// TIA Portal project "Project3_Sequence_Command" (V18)

(* hardware
DEVICE "S7-1500/ET200MP station_1"  S7-1500 station
   slot 0: "Rail_0"  Rack  6ES7 590-1***0-0AA0
DEVICE "S7-1500/ET200MP station_2"  S7-1500 station
   slot 0: "PM 190W 120/230VAC"  PM 190W 120/230VAC  6EP1333-4BA00
   slot 0: "Rail_0"  Rack  6ES7 590-1***0-0AA0
   slot 1: "PLC_1"  CPU 1516-3 PN/DP  6ES7 516-3AN01-0AB0  V2.1
      slot 3: "CPU display_1"  6ES7591-1BA00-0AA0
      slot 32768: "PROFINET interface_1"  X1
         slot 32769: "Port_1"  X1 P1
         slot 32770: "Port_2"  X1 P2
      slot 33024: "PROFINET interface_2"  X2
         slot 33025: "Port_1"  X2 P1
      slot 33280: "DP interface_1"  X3
   slot 2: "DI 32x24VDC HF_1"  DI 32x24VDC HF  6ES7 521-1BL00-0AB0  V2.2
   slot 3: "DQ 32x24VDC/0.5A HF_1"  DQ 32x24VDC/0.5A HF  6ES7 522-1BL01-0AB0  V1.1
   slot 4: "AI 8xU/R/RTD/TC HF_1"  AI 8xU/R/RTD/TC HF  6ES7 531-7PF00-0AB0  V1.1
   slot 5: "AQ 4xU/I HF_1"  AQ 4xU/I HF  6ES7 532-5ND00-0AB0  V1.1
*)

// ===== PLC "PLC_1"  CPU 1516-3 PN/DP =====

VAR_GLOBAL   // PLC tag table "Default tag table"
   "Tag_1" AT %I0.0 : Bool;
   "Tag_2" AT %Q0.0 : Bool;
   "Tag_3" AT %I0.1 : Bool;
   "Tag_4" AT %Q0.1 : Bool;
   "Tag_5" AT %M0.0 : Bool;
   "Tag_6" AT %Q0.2 : Bool;
   "Tag_7" AT %I0.2 : Bool;
   "Tag_8" AT %I0.3 : Bool;
   "Tag_9" AT %M1.0 : Bool;
   "Tag_10" AT %M1.1 : Bool;
   "Tag_11" AT %M0.1 : Bool;
   "Tag_12" AT %M0.2 : Bool;
   "Tag_13" AT %M1.2 : Bool;
   "Tag_14" AT %MD0 : Time;
   "Tag_15" AT %MD4 : Time;
   "Tag_16" AT %MD8 : Time;
   "Tag_17" AT %MD12 : Time;
   "Tag_18" AT %MD16 : Time;
   "Tag_19" AT %MW0 : Int;
   "Tag_20" AT %M1.3 : Bool;
   "Tag_21" AT %M2.0 : Bool;
END_VAR

// folder: System blocks/Program resources

DATA_BLOCK "DB1"   // DB1
{ S7_Optimized_Access := 'TRUE' }
AUTHOR : Simatic
FAMILY : IEC
NAME : IEC_TMR
VERSION : 1.0
// stored: InstanceOfName IEC_TIMER
"IEC_TIMER"
BEGIN
END_DATA_BLOCK

DATA_BLOCK "DB2"   // DB2
{ S7_Optimized_Access := 'TRUE' }
AUTHOR : Simatic
FAMILY : IEC
NAME : IEC_TMR
VERSION : 1.0
// stored: InstanceOfName IEC_TIMER
"IEC_TIMER"
BEGIN
END_DATA_BLOCK

DATA_BLOCK "DB3"   // DB3
{ S7_Optimized_Access := 'TRUE' }
AUTHOR : Simatic
FAMILY : IEC
NAME : IEC_TMR
VERSION : 1.0
// stored: InstanceOfName IEC_TIMER
"IEC_TIMER"
BEGIN
END_DATA_BLOCK

DATA_BLOCK "DB4"   // DB4
{ S7_Optimized_Access := 'TRUE' }
AUTHOR : Simatic
FAMILY : IEC
NAME : IEC_TMR
VERSION : 1.0
// stored: InstanceOfName IEC_TIMER
"IEC_TIMER"
BEGIN
END_DATA_BLOCK

DATA_BLOCK "DB5"   // DB5
{ S7_Optimized_Access := 'TRUE' }
AUTHOR : Simatic
FAMILY : IEC
NAME : IEC_TMR
VERSION : 1.0
// stored: InstanceOfName IEC_TIMER
"IEC_TIMER"
BEGIN
END_DATA_BLOCK

DATA_BLOCK "DB6"   // DB6
{ S7_Optimized_Access := 'TRUE' }
AUTHOR : Simatic
FAMILY : IEC
NAME : IEC_TMR
VERSION : 1.0
// stored: InstanceOfName IEC_TIMER
"IEC_TIMER"
BEGIN
END_DATA_BLOCK

DATA_BLOCK "DB7"   // DB7
{ S7_Optimized_Access := 'TRUE' }
AUTHOR : Simatic
FAMILY : IEC
NAME : IEC_TMR
VERSION : 1.0
// stored: InstanceOfName IEC_TIMER
"IEC_TIMER"
BEGIN
END_DATA_BLOCK

DATA_BLOCK "DB8"   // DB8
{ S7_Optimized_Access := 'TRUE' }
AUTHOR : Simatic
FAMILY : IEC
NAME : CNTR
VERSION : 1.0
// stored: InstanceOfName IEC_COUNTER
"IEC_COUNTER"
BEGIN
END_DATA_BLOCK

DATA_BLOCK "DB9"   // DB9
{ S7_Optimized_Access := 'TRUE' }
AUTHOR : Simatic
FAMILY : IEC
NAME : IEC_TMR
VERSION : 1.0
// stored: InstanceOfName IEC_TIMER
"IEC_TIMER"
BEGIN
END_DATA_BLOCK

DATA_BLOCK "DB10"   // DB10
{ S7_Optimized_Access := 'TRUE' }
AUTHOR : Simatic
FAMILY : IEC
NAME : IEC_TMR
VERSION : 1.0
// stored: InstanceOfName IEC_TIMER
"IEC_TIMER"
BEGIN
END_DATA_BLOCK

DATA_BLOCK "DB11"   // DB11
{ S7_Optimized_Access := 'TRUE' }
AUTHOR : Simatic
FAMILY : IEC
NAME : CNTR
VERSION : 1.0
// stored: InstanceOfName IEC_COUNTER
"IEC_COUNTER"
BEGIN
END_DATA_BLOCK

DATA_BLOCK "DB12"   // DB12
{ S7_Optimized_Access := 'TRUE' }
AUTHOR : Simatic
FAMILY : IEC
NAME : CNTR
VERSION : 1.0
// stored: InstanceOfName IEC_COUNTER
"IEC_COUNTER"
BEGIN
END_DATA_BLOCK

DATA_BLOCK "DB13"   // DB13
{ S7_Optimized_Access := 'TRUE' }
AUTHOR : Simatic
FAMILY : IEC
NAME : CNTR
VERSION : 1.0
// stored: InstanceOfName IEC_COUNTER
"IEC_COUNTER"
BEGIN
END_DATA_BLOCK

// folder: (top level)

ORGANIZATION_BLOCK "Main"   // OB1, LAD, ProgramCycle
TITLE = "Main Program Sweep (Cycle)"
{ S7_Optimized_Access := 'TRUE' }
VERSION : 0.1
   VAR_INPUT
      Initial_Call : Bool;   // Initial call of this OB
      Remanence : Bool;   // =True, if remanent data are available
   END_VAR
   VAR_TEMP   // added for the SCL form of the ladder/FBD networks
      _w1 : Bool;
      _w2 : Bool;
      _w3 : Bool;
   END_VAR
BEGIN

REGION Network 1: YES(긍정) 회로
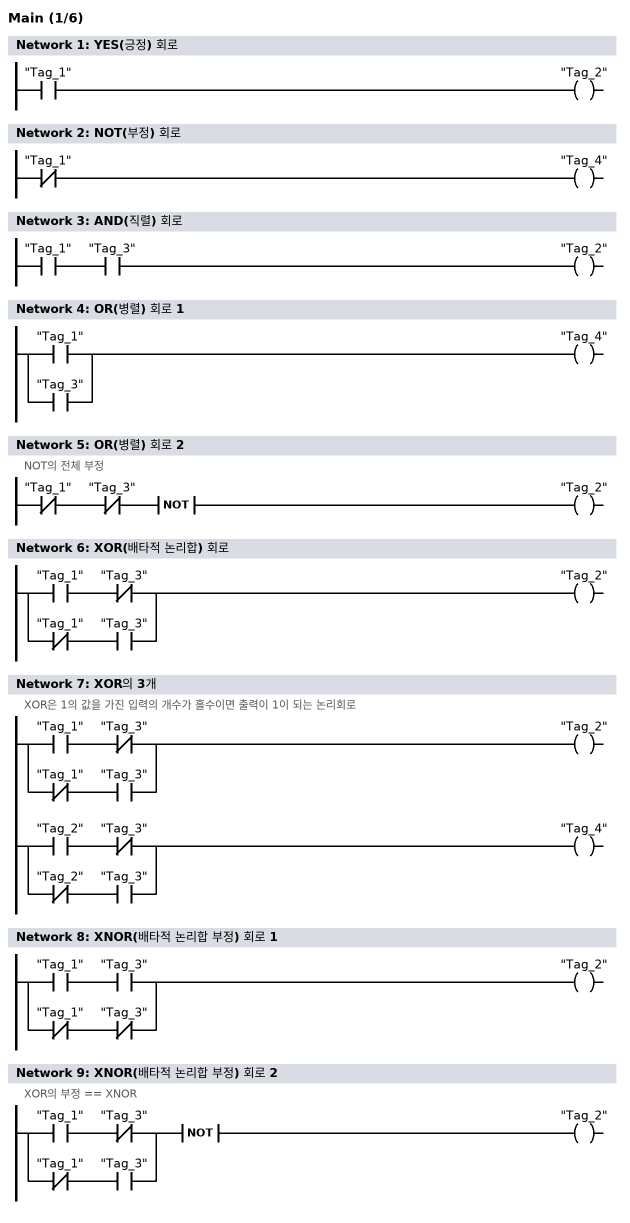
   RUNG wire#powerrail
      Contact( "Tag_1" )
      Coil( "Tag_2" )
   END_RUNG
   // the same network as SCL:
   "Tag_2" := "Tag_1";
END_REGION

REGION Network 2: NOT(부정) 회로
   RUNG wire#powerrail
      I_Contact( "Tag_1" )
      Coil( "Tag_4" )
   END_RUNG
   // the same network as SCL:
   "Tag_4" := NOT "Tag_1";
END_REGION

REGION Network 3: AND(직렬) 회로
   RUNG wire#powerrail
      Contact( "Tag_1" )
      Contact( "Tag_3" )
      Coil( "Tag_2" )
   END_RUNG
   // the same network as SCL:
   "Tag_2" := "Tag_1" AND "Tag_3";
END_REGION

REGION Network 4: OR(병렬) 회로 1
   RUNG wire#powerrail
      Contact( "Tag_1" )
      wire#w1
      Coil( "Tag_4" )
   END_RUNG
   RUNG wire#powerrail
      Contact( "Tag_3" )
   END_RUNG wire#w1
   // the same network as SCL:
   "Tag_4" := "Tag_1" OR "Tag_3";
END_REGION

REGION Network 5: OR(병렬) 회로 2
   // NOT의 전체 부정
   RUNG wire#powerrail
      I_Contact( "Tag_1" )
      I_Contact( "Tag_3" )
      Not()
      Coil( "Tag_2" )
   END_RUNG
   // the same network as SCL:
   "Tag_2" := NOT (NOT "Tag_1" AND NOT "Tag_3");
END_REGION

REGION Network 6: XOR(배타적 논리합) 회로
   RUNG wire#powerrail
      Contact( "Tag_1" )
      I_Contact( "Tag_3" )
      wire#w1
      Coil( "Tag_2" )
   END_RUNG
   RUNG wire#powerrail
      I_Contact( "Tag_1" )
      Contact( "Tag_3" )
   END_RUNG wire#w1
   // the same network as SCL:
   "Tag_2" := ("Tag_1" AND NOT "Tag_3") OR (NOT "Tag_1" AND "Tag_3");
END_REGION

REGION Network 7: XOR의 3개
   // XOR은 1의 값을 가진 입력의 개수가 홀수이면 출력이 1이 되는 논리회로
   RUNG wire#powerrail
      Contact( "Tag_1" )
      I_Contact( "Tag_3" )
      wire#w1
      Coil( "Tag_2" )
   END_RUNG
   RUNG wire#powerrail
      I_Contact( "Tag_1" )
      Contact( "Tag_3" )
   END_RUNG wire#w1
   RUNG wire#powerrail
      Contact( "Tag_2" )
      I_Contact( "Tag_3" )
      wire#w2
      Coil( "Tag_4" )
   END_RUNG
   RUNG wire#powerrail
      I_Contact( "Tag_2" )
      Contact( "Tag_3" )
   END_RUNG wire#w2
   // the same network as SCL:
   "Tag_2" := ("Tag_1" AND NOT "Tag_3") OR (NOT "Tag_1" AND "Tag_3");
   "Tag_4" := ("Tag_2" AND NOT "Tag_3") OR (NOT "Tag_2" AND "Tag_3");
END_REGION

REGION Network 8: XNOR(배타적 논리합 부정) 회로 1
   RUNG wire#powerrail
      Contact( "Tag_1" )
      Contact( "Tag_3" )
      wire#w1
      Coil( "Tag_2" )
   END_RUNG
   RUNG wire#powerrail
      I_Contact( "Tag_1" )
      I_Contact( "Tag_3" )
   END_RUNG wire#w1
   // the same network as SCL:
   "Tag_2" := ("Tag_1" AND "Tag_3") OR (NOT "Tag_1" AND NOT "Tag_3");
END_REGION

REGION Network 9: XNOR(배타적 논리합 부정) 회로 2
   // XOR의 부정 == XNOR
   RUNG wire#powerrail
      Contact( "Tag_1" )
      I_Contact( "Tag_3" )
      wire#w1
      Not()
      Coil( "Tag_2" )
   END_RUNG
   RUNG wire#powerrail
      I_Contact( "Tag_1" )
      Contact( "Tag_3" )
   END_RUNG wire#w1
   // the same network as SCL:
   "Tag_2" := NOT (("Tag_1" AND NOT "Tag_3") OR (NOT "Tag_1" AND "Tag_3"));
END_REGION

REGION Network 10: 자기유지 회로 1 - 리셋 우선 자기유지 회로
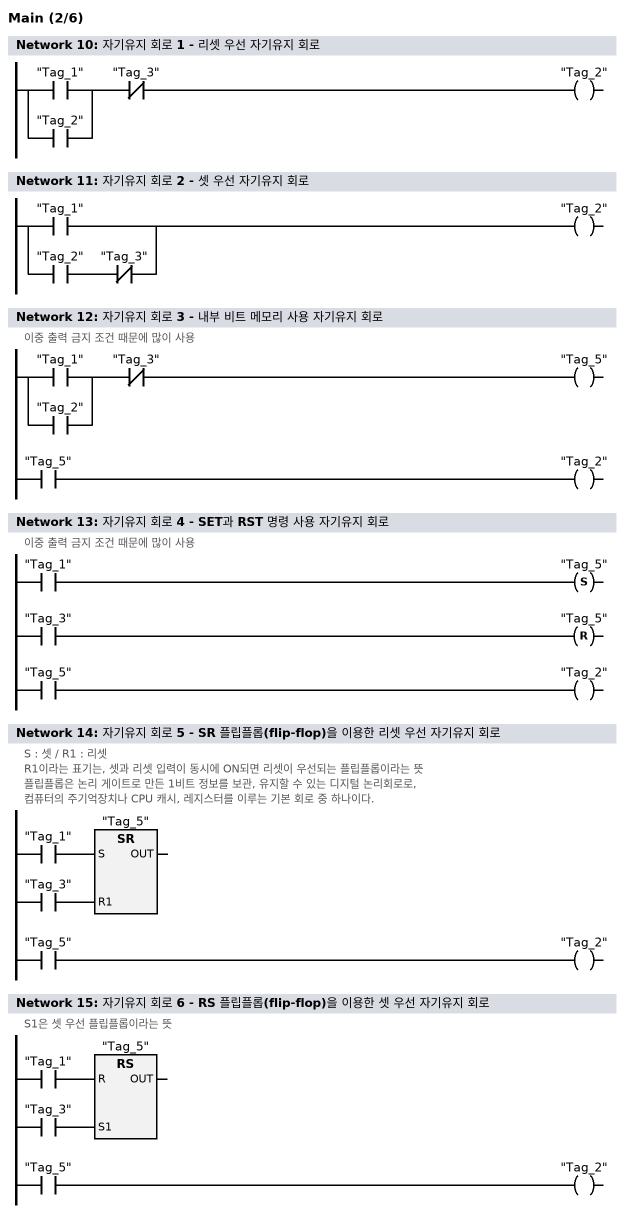
   RUNG wire#powerrail
      Contact( "Tag_1" )
      wire#w1
      I_Contact( "Tag_3" )
      Coil( "Tag_2" )
   END_RUNG
   RUNG wire#powerrail
      Contact( "Tag_2" )
   END_RUNG wire#w1
   // the same network as SCL:
   "Tag_2" := ("Tag_1" OR "Tag_2") AND NOT "Tag_3";
END_REGION

REGION Network 11: 자기유지 회로 2 - 셋 우선 자기유지 회로
   RUNG wire#powerrail
      Contact( "Tag_1" )
      wire#w1
      Coil( "Tag_2" )
   END_RUNG
   RUNG wire#powerrail
      Contact( "Tag_2" )
      I_Contact( "Tag_3" )
   END_RUNG wire#w1
   // the same network as SCL:
   "Tag_2" := "Tag_1" OR ("Tag_2" AND NOT "Tag_3");
END_REGION

REGION Network 12: 자기유지 회로 3 - 내부 비트 메모리 사용 자기유지 회로
   // 이중 출력 금지 조건 때문에 많이 사용
   RUNG wire#powerrail
      Contact( "Tag_1" )
      wire#w1
      I_Contact( "Tag_3" )
      Coil( "Tag_5" )
   END_RUNG
   RUNG wire#powerrail
      Contact( "Tag_2" )
   END_RUNG wire#w1
   RUNG wire#powerrail
      Contact( "Tag_5" )
      Coil( "Tag_2" )
   END_RUNG
   // the same network as SCL:
   "Tag_5" := ("Tag_1" OR "Tag_2") AND NOT "Tag_3";
   "Tag_2" := "Tag_5";
END_REGION

REGION Network 13: 자기유지 회로 4 - SET과 RST 명령 사용 자기유지 회로
   // 이중 출력 금지 조건 때문에 많이 사용
   RUNG wire#powerrail
      Contact( "Tag_1" )
      S_Coil( "Tag_5" )
   END_RUNG
   RUNG wire#powerrail
      Contact( "Tag_3" )
      R_Coil( "Tag_5" )
   END_RUNG
   RUNG wire#powerrail
      Contact( "Tag_5" )
      Coil( "Tag_2" )
   END_RUNG
   // the same network as SCL:
   IF "Tag_1" THEN "Tag_5" := TRUE; END_IF;
   IF "Tag_3" THEN "Tag_5" := FALSE; END_IF;
   "Tag_2" := "Tag_5";
END_REGION

REGION Network 14: 자기유지 회로 5 - SR 플립플롭(flip-flop)을 이용한 리셋 우선 자기유지 회로
   // S : 셋 / R1 : 리셋
   // 
   // R1이라는 표기는, 셋과 리셋 입력이 동시에 ON되면 리셋이 우선되는 플립플롭이라는 뜻
   // 
   // 플립플롭은 논리 게이트로 만든 1비트 정보를 보관, 유지할 수 있는 디지털 논리회로로,
   // 컴퓨터의 주기억장치나 CPU 캐시, 레지스터를 이루는 기본 회로 중 하나이다.
   RUNG wire#powerrail
      Contact( "Tag_1" )
      S_SR(operand := "Tag_5", r1 := wire#w1)
   END_RUNG
   RUNG wire#powerrail
      Contact( "Tag_3" )
   END_RUNG wire#w1
   RUNG wire#powerrail
      Contact( "Tag_5" )
      Coil( "Tag_2" )
   END_RUNG
   // the same network as SCL:
   IF "Tag_1" THEN
       "Tag_5" := TRUE;   // SR flip-flop
   END_IF;
   IF "Tag_3" THEN "Tag_5" := FALSE; END_IF;
   "Tag_2" := "Tag_5";
END_REGION

REGION Network 15: 자기유지 회로 6 - RS 플립플롭(flip-flop)을 이용한 셋 우선 자기유지 회로
   // S1은 셋 우선 플립플롭이라는 뜻
   RUNG wire#powerrail
      Contact( "Tag_1" )
      S_RS(operand := "Tag_5", s1 := wire#w1)
   END_RUNG
   RUNG wire#powerrail
      Contact( "Tag_3" )
   END_RUNG wire#w1
   RUNG wire#powerrail
      Contact( "Tag_5" )
      Coil( "Tag_2" )
   END_RUNG
   // the same network as SCL:
   IF "Tag_1" THEN
       "Tag_5" := FALSE;   // RS flip-flop
   END_IF;
   IF "Tag_3" THEN "Tag_5" := TRUE; END_IF;
   "Tag_2" := "Tag_5";
END_REGION

REGION Network 16: 자기유지 회로 7(선입 우선회로) - 리셋 우선 자기유지 회로를 사용한 선입 우선회로
   // 선입 우선회로는 현재 실행되고 있는 작업이 있을 경우에 다른 작업의 실행을 거부하는 전기회로
   // 
   // 선입 우선회로는 먼저 입력된 정보를 기억하고, 다른 정보의 입력을 막는 역할을 하는 전기회로를 의미
   // ex) 퀴즈쇼 램프 버튼
   // 
   // → 선입 우선회로는 '리셋 우선 자기유지' 회로로 구성된다.
   // 
   // 
   // I0.0 : 리셋 푸시버튼
   // I0.1 : 출연자1 푸시버튼
   // I0.2 : 출연자2 푸시버튼
   // I0.3 : 출연자3 푸시버튼
   // Q0.0 : 출연자1 램프
   // Q0.1 : 출연자2 램프
   // Q0.2 : 출연자3 램프
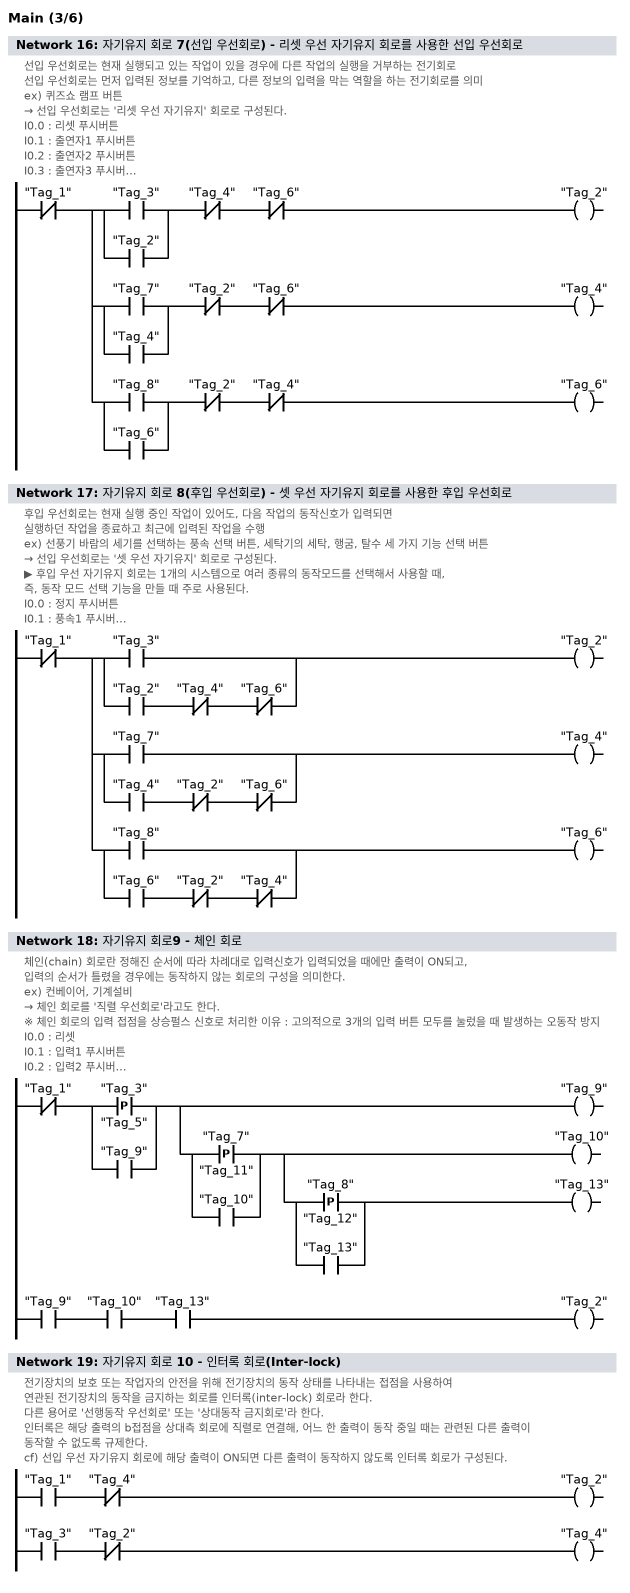
   RUNG wire#powerrail
      I_Contact( "Tag_1" )
      wire#w1
      Contact( "Tag_3" )
      wire#w2
      I_Contact( "Tag_4" )
      I_Contact( "Tag_6" )
      Coil( "Tag_2" )
   END_RUNG
   RUNG wire#w1
      Contact( "Tag_2" )
   END_RUNG wire#w2
   RUNG wire#w1
      Contact( "Tag_7" )
      wire#w3
      I_Contact( "Tag_2" )
      I_Contact( "Tag_6" )
      Coil( "Tag_4" )
   END_RUNG
   RUNG wire#w1
      Contact( "Tag_4" )
   END_RUNG wire#w3
   RUNG wire#w1
      Contact( "Tag_8" )
      wire#w4
      I_Contact( "Tag_2" )
      I_Contact( "Tag_4" )
      Coil( "Tag_6" )
   END_RUNG
   RUNG wire#w1
      Contact( "Tag_6" )
   END_RUNG wire#w4
   // the same network as SCL:
   "Tag_2" := NOT "Tag_1" AND ("Tag_3" OR "Tag_2") AND NOT "Tag_4" AND NOT "Tag_6";
   "Tag_4" := NOT "Tag_1" AND ("Tag_7" OR "Tag_4") AND NOT "Tag_2" AND NOT "Tag_6";
   "Tag_6" := NOT "Tag_1" AND ("Tag_8" OR "Tag_6") AND NOT "Tag_2" AND NOT "Tag_4";
END_REGION

REGION Network 17: 자기유지 회로 8(후입 우선회로) - 셋 우선 자기유지 회로를 사용한 후입 우선회로
   // 후입 우선회로는 현재 실행 중인 작업이 있어도, 다음 작업의 동작신호가 입력되면 
   // 실행하던 작업을 종료하고 최근에 입력된 작업을 수행
   // ex) 선풍기 바람의 세기를 선택하는 풍속 선택 버튼, 세탁기의 세탁, 행굼, 탈수 세 가지 기능 선택 버튼
   // 
   // → 선입 우선회로는 '셋 우선 자기유지' 회로로 구성된다.
   // ▶ 후입 우선 자기유지 회로는 1개의 시스템으로 여러 종류의 동작모드를 선택해서 사용할 때,
   // 즉, 동작 모드 선택 기능을 만들 때 주로 사용된다.
   // 
   // 
   // I0.0 : 정지 푸시버튼
   // I0.1 : 풍속1 푸시버튼
   // I0.2 : 풍속2 푸시버튼
   // I0.3 : 풍속3 푸시버튼
   // Q0.0 : 풍속1 램프
   // Q0.1 : 풍속2 램프
   // Q0.2 : 풍속3 램프
   RUNG wire#powerrail
      I_Contact( "Tag_1" )
      wire#w1
      Contact( "Tag_3" )
      wire#w2
      Coil( "Tag_2" )
   END_RUNG
   RUNG wire#w1
      Contact( "Tag_2" )
      I_Contact( "Tag_4" )
      I_Contact( "Tag_6" )
   END_RUNG wire#w2
   RUNG wire#w1
      Contact( "Tag_7" )
      wire#w3
      Coil( "Tag_4" )
   END_RUNG
   RUNG wire#w1
      Contact( "Tag_4" )
      I_Contact( "Tag_2" )
      I_Contact( "Tag_6" )
   END_RUNG wire#w3
   RUNG wire#w1
      Contact( "Tag_8" )
      wire#w4
      Coil( "Tag_6" )
   END_RUNG
   RUNG wire#w1
      Contact( "Tag_6" )
      I_Contact( "Tag_2" )
      I_Contact( "Tag_4" )
   END_RUNG wire#w4
   // the same network as SCL:
   "Tag_2" := NOT "Tag_1" AND ("Tag_3" OR ("Tag_2" AND NOT "Tag_4" AND NOT "Tag_6"));
   "Tag_4" := NOT "Tag_1" AND ("Tag_7" OR ("Tag_4" AND NOT "Tag_2" AND NOT "Tag_6"));
   "Tag_6" := NOT "Tag_1" AND ("Tag_8" OR ("Tag_6" AND NOT "Tag_2" AND NOT "Tag_4"));
END_REGION

REGION Network 18: 자기유지 회로9 - 체인 회로
   // 체인(chain) 회로란 정해진 순서에 따라 차례대로 입력신호가 입력되었을 때에만 출력이 ON되고,
   // 입력의 순서가 틀렸을 경우에는 동작하지 않는 회로의 구성을 의미한다.
   // ex) 컨베이어, 기계설비
   // 
   // → 체인 회로를 '직렬 우선회로'라고도 한다.
   // 
   // ※ 체인 회로의 입력 접점을 상승펄스 신호로 처리한 이유 : 고의적으로 3개의 입력 버튼 모두를 눌렀을 때 발생하는 오동작 방지
   // 
   // 
   // I0.0 : 리셋
   // I0.1 : 입력1 푸시버튼
   // I0.2 : 입력2 푸시버튼
   // I0.3 : 입력3 푸시버튼
   // Q0.0 : 선택 램프
   RUNG wire#powerrail
      I_Contact( "Tag_1" )
      wire#w1
      P_Contact(operand := "Tag_3", bit := "Tag_5")
      wire#w2
      Coil( "Tag_9" )
   END_RUNG
   RUNG wire#w1
      Contact( "Tag_9" )
   END_RUNG wire#w2
   RUNG wire#w2
      P_Contact(operand := "Tag_7", bit := "Tag_11")
      wire#w3
      Coil( "Tag_10" )
   END_RUNG
   RUNG wire#w2
      Contact( "Tag_10" )
   END_RUNG wire#w3
   RUNG wire#w3
      P_Contact(operand := "Tag_8", bit := "Tag_12")
      wire#w4
      Coil( "Tag_13" )
   END_RUNG
   RUNG wire#w3
      Contact( "Tag_13" )
   END_RUNG wire#w4
   RUNG wire#powerrail
      Contact( "Tag_9" )
      Contact( "Tag_10" )
      Contact( "Tag_13" )
      Coil( "Tag_2" )
   END_RUNG
   // the same network as SCL:
   #_w1 := NOT "Tag_1" AND "Tag_3" AND NOT "Tag_5";   // rising edge of "Tag_3"
   "Tag_5" := "Tag_3";
   "Tag_9" := #_w1 OR (NOT "Tag_1" AND "Tag_9");
   #_w2 := "Tag_9" AND "Tag_7" AND NOT "Tag_11";   // rising edge of "Tag_7"
   "Tag_11" := "Tag_7";
   "Tag_10" := #_w2 OR ("Tag_9" AND "Tag_10");
   #_w3 := "Tag_10" AND "Tag_8" AND NOT "Tag_12";   // rising edge of "Tag_8"
   "Tag_12" := "Tag_8";
   "Tag_13" := #_w3 OR ("Tag_10" AND "Tag_13");
   "Tag_2" := "Tag_9" AND "Tag_10" AND "Tag_13";
END_REGION

REGION Network 19: 자기유지 회로 10 - 인터록 회로(Inter-lock)
   // 전기장치의 보호 또는 작업자의 안전을 위해 전기장치의 동작 상태를 나타내는 접점을 사용하여
   // 연관된 전기장치의 동작을 금지하는 회로를 인터록(inter-lock) 회로라 한다.
   // 다른 용어로 '선행동작 우선회로' 또는 '상대동작 금지회로'라 한다.
   // 인터록은 해당 출력의 b접점을 상대측 회로에 직렬로 연결해, 어느 한 출력이 동작 중일 때는 관련된 다른 출력이
   // 동작할 수 없도록 규제한다.
   // 
   // cf) 선입 우선 자기유지 회로에 해당 출력이 ON되면 다른 출력이 동작하지 않도록 인터록 회로가 구성된다.
   RUNG wire#powerrail
      Contact( "Tag_1" )
      I_Contact( "Tag_4" )
      Coil( "Tag_2" )
   END_RUNG
   RUNG wire#powerrail
      Contact( "Tag_3" )
      I_Contact( "Tag_2" )
      Coil( "Tag_4" )
   END_RUNG
   // the same network as SCL:
   "Tag_2" := "Tag_1" AND NOT "Tag_4";
   "Tag_4" := "Tag_3" AND NOT "Tag_2";
END_REGION

REGION Network 20: 타이머 회로 1 - TON(온 딜레이 타이머)
   // 입력이 ON되면 사전 설정된 시간(PT)이 경과한 후에 타이머의 출력이 ON되고,
   // 입력이 OFF되면 출력도 함께 OFF된다.
   // 
   // PT : Preset Time - 설정 시간
   // ET : Elapsed Time - 현재 시간(경과 시간)
   // PT 및 ET의 태그 타입은 TIME
   // TIME은 32비트를 사용하기 때문에 MD의 메모리 설정
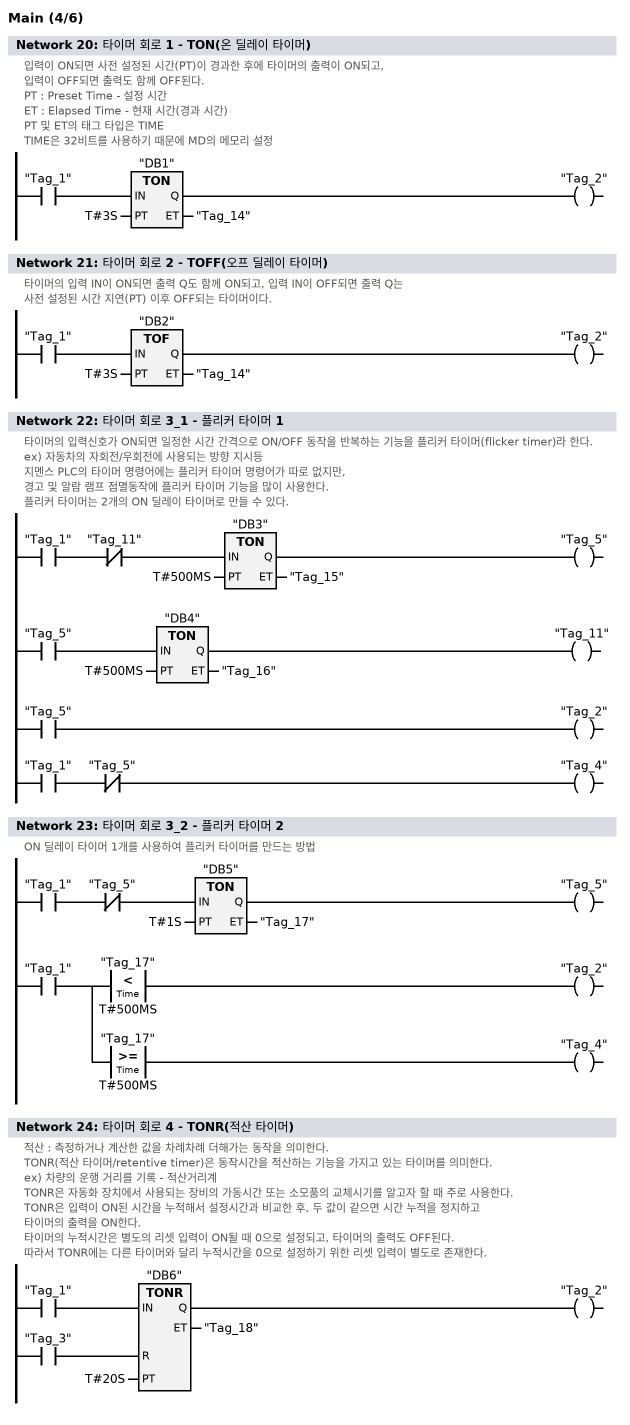
   "DB1".TON(IN := "Tag_1", PT := T#3S, ET => "Tag_14");
   "Tag_2" := "DB1".Q;
END_REGION

REGION Network 21: 타이머 회로 2 - TOFF(오프 딜레이 타이머)
   // 타이머의 입력 IN이 ON되면 출력 Q도 함께 ON되고, 입력 IN이 OFF되면 출력 Q는
   // 사전 설정된 시간 지연(PT) 이후 OFF되는 타이머이다.
   "DB2".TOF(IN := "Tag_1", PT := T#3S, ET => "Tag_14");
   "Tag_2" := "DB2".Q;
END_REGION

REGION Network 22: 타이머 회로 3_1 - 플리커 타이머 1
   // 타이머의 입력신호가 ON되면 일정한 시간 간격으로 ON/OFF 동작을 반복하는 기능을 플리커 타이머(flicker timer)라 한다.
   // ex) 자동차의 자회전/우회전에 사용되는 방향 지시등
   // 
   // 지멘스 PLC의 타이머 명령어에는 플리커 타이머 명령어가 따로 없지만,
   // 경고 및 알람 램프 점멸동작에 플리커 타이머 기능을 많이 사용한다.
   // 
   // 플리커 타이머는 2개의 ON 딜레이 타이머로 만들 수 있다.
   "DB3".TON(IN := "Tag_1" AND NOT "Tag_11", PT := T#500MS, ET => "Tag_15");
   "Tag_5" := "DB3".Q;
   "DB4".TON(IN := "Tag_5", PT := T#500MS, ET => "Tag_16");
   "Tag_11" := "DB4".Q;
   "Tag_2" := "Tag_5";
   "Tag_4" := "Tag_1" AND NOT "Tag_5";
END_REGION

REGION Network 23: 타이머 회로 3_2 - 플리커 타이머 2
   // ON 딜레이 타이머 1개를 사용하여 플리커 타이머를 만드는 방법
   "DB5".TON(IN := "Tag_1" AND NOT "Tag_5", PT := T#1S, ET => "Tag_17");
   "Tag_5" := "DB5".Q;
   "Tag_2" := "Tag_1" AND ("Tag_17" < T#500MS);
   "Tag_4" := "Tag_1" AND ("Tag_17" >= T#500MS);
END_REGION

REGION Network 24: 타이머 회로 4 - TONR(적산 타이머)
   // 적산 : 측정하거나 계산한 값을 차례차례 더해가는 동작을 의미한다.
   // TONR(적산 타이머/retentive timer)은 동작시간을 적산하는 기능을 가지고 있는 타이머를 의미한다.
   // ex) 차량의 운행 거리를 기록 - 적산거리계
   // 
   // TONR은 자동화 장치에서 사용되는 장비의 가동시간 또는 소모품의 교체시기를 알고자 할 때 주로 사용한다.
   // TONR은 입력이 ON된 시간을 누적해서 설정시간과 비교한 후, 두 값이 같으면 시간 누적을 정지하고
   // 타이머의 출력을 ON한다.
   // 타이머의 누적시간은 별도의 리셋 입력이 ON될 때 0으로 설정되고, 타이머의 출력도 OFF된다.
   // 따라서 TONR에는 다른 타이머와 달리 누적시간을 0으로 설정하기 위한 리셋 입력이 별도로 존재한다.
   "DB6".TONR(IN := "Tag_1", R := "Tag_3", PT := T#20S, ET => "Tag_18");
   "Tag_2" := "DB6".Q;
END_REGION

REGION Network 25: 타이머 회로 5_1 - TP(펄스 타이머) - ON 후 펄스신호 출력
   // 타이머 설정시간 PT에 관계없이 입력만 ON되면 일정한 시간 동안 타이머의 출력이 ON되는 타이머이다.
   // 
   // a접점 신호를 사용하면, IN 입력신호가 ON된 시간에 관계없이 출력은 PT 입력에 설정된 시간만큼 ON된다.
   // 
   // 입력신호의 시간에 관계없이 입력신호가 ON되면 출력이 정해진 일정시간 동안 ON되는 TP 동작을 
   // '원 샷 타이머(one shot timer)'라 부르기도 한다.
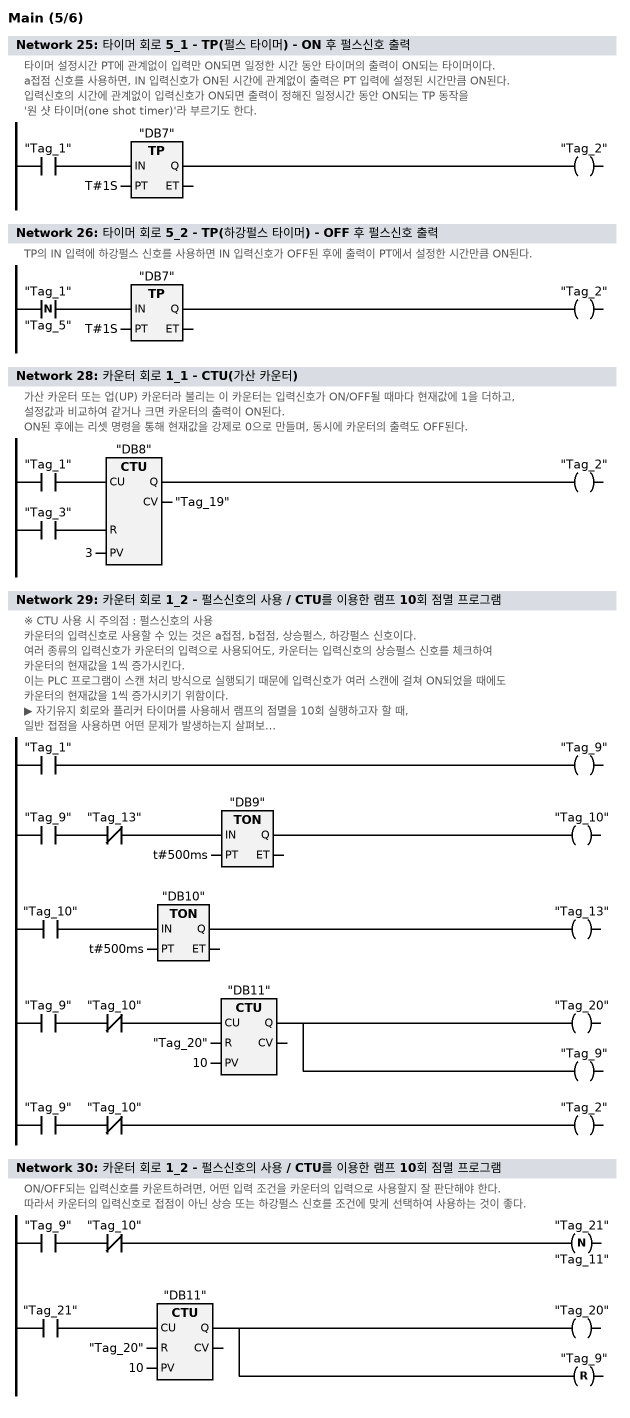
   "DB7".TP(IN := "Tag_1", PT := T#1S);
   "Tag_2" := "DB7".Q;
END_REGION

REGION Network 26: 타이머 회로 5_2 - TP(하강펄스 타이머) - OFF 후 펄스신호 출력
   // TP의 IN 입력에 하강펄스 신호를 사용하면 IN 입력신호가 OFF된 후에 출력이 PT에서 설정한 시간만큼 ON된다.
   #_w1 := NOT "Tag_1" AND "Tag_5";   // falling edge of "Tag_1"
   "Tag_5" := "Tag_1";
   "DB7".TP(IN := #_w1, PT := T#1S);
   "Tag_2" := "DB7".Q;
END_REGION

REGION Network 27: 카운터 회로
   // 카운터(Counter)는 '수를 세는 장치'라는 의미
   // 전기 스위치의 ON/OFF 횟수를 세거나, 센서의 ON/OFF 신호를 세는 역할을 한다.
   // 
   // 지멘스 PLC S7-300/1500에서는 타이머와 비슷하게 S5 PLC부터 사용하던 카운터와 IEC 카운터 명령어로 구분한다.
   // (여기서는 IEC 카운터만 설명)
   // 
   // IEC 카운터는 동작 기능에 따라 가산 카운터(CTU)와 감산 카운터(CTD), 가감산 카운터(CTUD)로 구분된다.
END_REGION

REGION Network 28: 카운터 회로 1_1 - CTU(가산 카운터)
   // 가산 카운터 또는 업(UP) 카운터라 불리는 이 카운터는 입력신호가 ON/OFF될 때마다 현재값에 1을 더하고,
   // 설정값과 비교하여 같거나 크면 카운터의 출력이 ON된다.
   // ON된 후에는 리셋 명령을 통해 현재값을 강제로 0으로 만들며, 동시에 카운터의 출력도 OFF된다.
   "DB8".CTU(CU := "Tag_1", R := "Tag_3", PV := 3, CV => "Tag_19");
   "Tag_2" := "DB8".Q;
END_REGION

REGION Network 29: 카운터 회로 1_2 - 펄스신호의 사용 / CTU를 이용한 램프 10회 점멸 프로그램
   // ※ CTU 사용 시 주의점 : 펄스신호의 사용
   // 
   // 카운터의 입력신호로 사용할 수 있는 것은 a접점, b접점, 상승펄스, 하강펄스 신호이다.
   // 여러 종류의 입력신호가 카운터의 입력으로 사용되어도, 카운터는 입력신호의 상승펄스 신호를 체크하여
   // 카운터의 현재값을 1씩 증가시킨다.
   // 이는 PLC 프로그램이 스캔 처리 방식으로 실행되기 때문에 입력신호가 여러 스캔에 걸쳐 ON되었을 때에도
   // 카운터의 현재값을 1씩 증가시키기 위함이다.
   // 
   // ▶ 자기유지 회로와 플리커 타이머를 사용해서 램프의 점멸을 10회 실행하고자 할 때,
   //     일반 접점을 사용하면 어떤 문제가 발생하는지 살펴보기
   // 
   // ● 첫 번째 프로그램 라인은 I0.0의 버튼을 누르면 M1.0의 비트 메모리 값을 1로 설정하는 동작
   // ● 두 번째와 세 번째 프로그램은 주기가 1sec(500ms ON, 500ms OFF)인 플리커 타이머 동작
   // ● 네 번째 라인에서는 플리커 타이머에 의해 ON되는 펄스신호를 가산 타이머를 사용해서 카운팅
   //     (가산 카운터의 PV의 설정값과 같아지면 가산 카운터의 출력 Q가 ON)
   // ● 비트가 리셋되면 두 번째 프로그램 라인의 M1.0도 OFF되어 플리커 타이머의 동작을 중지시킨다.
   //     이때 가산 카운터도 자신의 출력으로 스스로를 리셋한다.
   // 
   // ◇ 카운터는 입력신호의 상승펄스에서 카운터의 값을 증가시킨다. 따라서 상승펄스신호가 10번째 입력되는 순간, 
   //      플리커 타이머의 동작이 중지되면서 램프가 9회만 점등된다.
   // ◇ 램프의 점멸을 10회 반복하려면 입력신호를 하강펄스로 변경하면 된다. (아래 참조)
   "Tag_9" := "Tag_1";
   "DB9".TON(IN := "Tag_9" AND NOT "Tag_13", PT := t#500ms);
   "Tag_10" := "DB9".Q;
   "DB10".TON(IN := "Tag_10", PT := t#500ms);
   "Tag_13" := "DB10".Q;
   "DB11".CTU(CU := "Tag_9" AND NOT "Tag_10", R := "Tag_20", PV := 10);
   "Tag_20" := "DB11".Q;
   "Tag_9" := "DB11".Q;
   "Tag_2" := "Tag_9" AND NOT "Tag_10";
END_REGION

REGION Network 30: 카운터 회로 1_2 - 펄스신호의 사용 / CTU를 이용한 램프 10회 점멸 프로그램
   // ON/OFF되는 입력신호를 카운트하려면, 어떤 입력 조건을 카운터의 입력으로 사용할지 잘 판단해야 한다.
   // 따라서 카운터의 입력신호로 접점이 아닌 상승 또는 하강펄스 신호를 조건에 맞게 선택하여 사용하는 것이 좋다.
   #_w1 := "Tag_9" AND NOT "Tag_10";
   "Tag_21" := NOT #_w1 AND "Tag_11";   // falling edge
   "Tag_11" := #_w1;
   "DB11".CTU(CU := "Tag_21", R := "Tag_20", PV := 10);
   "Tag_20" := "DB11".Q;
   IF "DB11".Q THEN "Tag_9" := FALSE; END_IF;
END_REGION

REGION Network 31: 카운터 회로 2 - CTD(감산 카운터)
   // 감산 카운터 또는 다운(DOWN) 카운터라 불리는 이 카운터는 입력신호가 ON/OFF될 때마다 설정된
   // 현재값에서 1씩 감산하다가, 현재값이 0과 같거나 작으면 카운터의 출력을 ON시킨다.
   // 출력이 ON된 후 LD 입력을 ON하면, PV에 설정된 값이 CV로 전송되면서 CV의 값이 0보다 크게 설정되기 때문에
   // 출력이 OFF 된다.
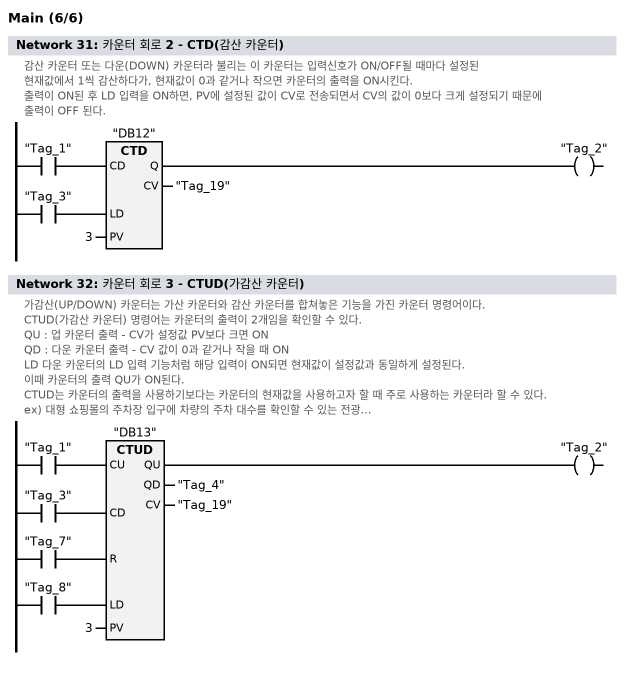
   "DB12".CTD(CD := "Tag_1", LD := "Tag_3", PV := 3, CV => "Tag_19");
   "Tag_2" := "DB12".Q;
END_REGION

REGION Network 32: 카운터 회로 3 - CTUD(가감산 카운터)
   // 가감산(UP/DOWN) 카운터는 가산 카운터와 감산 카운터를 합쳐놓은 기능을 가진 카운터 명령어이다.
   // CTUD(가감산 카운터) 명령어는 카운터의 출력이 2개임을 확인할 수 있다.
   // QU : 업 카운터 출력 - CV가 설정값 PV보다 크면 ON
   // QD : 다운 카운터 출력 - CV 값이 0과 같거나 작을 때 ON 
   // 
   // LD 다운 카운터의 LD 입력 기능처럼 해당 입력이 ON되면 현재값이 설정값과 동일하게 설정된다.
   // 이때 카운터의 출력 QU가 ON된다.
   // 
   // CTUD는 카운터의 출력을 사용하기보다는 카운터의 현재값을 사용하고자 할 때 주로 사용하는 카운터라 할 수 있다.
   // ex) 대형 쇼핑몰의 주차장 입구에 차량의 주차 대수를 확인할 수 있는 전광판
   //       ● 차량 입고 검출 센서 카운터 업(증가) - %I0.0
   //       ● 차량 출고 검출 센서 카운터 다운(감소) - %I0.1
   //       ● 만차 표시 램프 - %Q0.0
   //       ● 주차 표시 램프 - %Q0.1
   "DB13".CTUD(CU := "Tag_1",
               CD := "Tag_3",
               R := "Tag_7",
               LD := "Tag_8",
               PV := 3,
               QD => "Tag_4",
               CV => "Tag_19");
   "Tag_2" := "DB13".QU;
END_REGION
END_ORGANIZATION_BLOCK